(*~
	<docu>
		<summary>
			Provides dialog with the user to allow for deciding how to proceed in case of failure.	
		</summary>	
	</docu>	
~*)
FUNCTION_BLOCK PUBLIC TcoInspectorDialog EXTENDS TcoCore.TcoDialogBase
VAR
    _dialogRetry : BOOL;
    _dialogTerminate : BOOL;
    _dialogOverride : BOOL;
    _dialogIsClosed : BOOL;
    _isOverInspected : BOOL;
    {attribute 'hide'}
    _refInspector : REFERENCE TO TcoInspector;
    {attribute 'hide'}
    _tierAct : TcoCore.TcoTier(THIS^);

    _rTrigRetry : R_TRIG;
    _rTrigTerminate : R_TRIG;
    _externalCloseReq : BOOL;
    _closeRetrySignal : BOOL;
    _closeTerminateSignal : BOOL;

    _instruction : STRING(255);
    _source : STRING(255);
    _imageHeight : REAL;
    _imageWidth : REAL;
    _hideOverideButton : BOOL;
    _hideTerminateButton : BOOL;
    _hideRetryButton : BOOL;

    _showFailureDescription : BOOL;
    _showErrorCode : BOOL;
    _showDescription : BOOL;

    _isInvoked : BOOL;
END_VAR

SUPER^();

PROPERTY DialogIsClosed: REFERENCE TO BOOL
GET
DialogIsClosed ref=_dialogIsClosed;
END_GET
END_PROPERTY

PROPERTY DialogOverride: REFERENCE TO BOOL
GET
DialogOverride ref=_dialogOverride;
END_GET
END_PROPERTY

PROPERTY DialogRetry: REFERENCE TO BOOL
GET
DialogRetry ref=_dialogRetry;
END_GET
END_PROPERTY

PROPERTY DialogTerminate: REFERENCE TO BOOL
GET
DialogTerminate ref=_dialogTerminate;
END_GET
END_PROPERTY

{attribute 'hide'}
METHOD PUBLIC FB_init : BOOL
VAR_INPUT
	bInitRetains : BOOL; // if TRUE, the retain variables are initialized (warm start / cold start)
	bInCopyCode : BOOL;  // if TRUE, the instance afterwards gets moved into the copy code (online change)
	ParentObject : ITcoObject;
END_VAR
END_METHOD

METHOD HandleExternalSignals
VAR_INPUT
	inRetrySignal:BOOL;
	inTerminateSignal : BOOL;
	
END_VAR

_closeRetrySignal:=FALSE;
_closeTerminateSignal:=FALSE;


_rTrigRetry(CLK:=inRetrySignal);
IF _rTrigRetry.q THEN
	_closeRetrySignal:=TRUE;
END_IF

_rTrigTerminate(CLK:=inTerminateSignal);
IF _rTrigTerminate.q THEN
	_closeTerminateSignal:=TRUE;
END_IF

 IF(_refInspector.Done) THEN	
	 	IF NOT ( _dialogRetry) THEN
			_dialogRetry:=_closeRetrySignal;
		END_IF;
		IF NOT ( _dialogTerminate) THEN
			_dialogTerminate:=_closeTerminateSignal;
		END_IF;
 END_IF
END_METHOD

PROPERTY HideOverride: REFERENCE TO BOOL
GET
HideOverride ref=_hideOverideButton;
END_GET
END_PROPERTY

PROPERTY HideRetry: REFERENCE TO BOOL
GET
HideRetry ref=_hideRetryButton;
END_GET
END_PROPERTY

PROPERTY HideTetminate: REFERENCE TO BOOL
GET
HideTetminate ref=_hideTerminateButton;
END_GET
END_PROPERTY

METHOD PROTECTED OnStart
SUPER^.OnStart();
_isInvoked:=TRUE;
_dialogIsClosed:=FALSE;
_dialogRetry	    :=  FALSE;	
_dialogTerminate  	:=  FALSE;	
_dialogOverride   	:=  FALSE;
END_METHOD

PROPERTY INTERNAL OverInspected : BOOL
GET
OverInspected := _isOverInspected;
END_GET
SET
_isOverInspected := OverInspected;
END_SET
END_PROPERTY

METHOD Restore : TcoCore.ITcoRestorable
VAR_INPUT
END_VAR
SUPER^.Restore();
_dialogRetry	    :=  FALSE;	
_dialogTerminate  	:=  FALSE;	
_dialogOverride   	:=  FALSE;

_instruction:='';
_source:='';
_hideOverideButton:=FALSE;
_hideRetryButton:=FALSE;
_hideTerminateButton:=FALSE;
_imageHeight:=400;
_imageWidth:=600;
_showDescription:=FALSE;
_showFailureDescription:=FALSE;
_showErrorCode:=FALSE;
_isInvoked:=FALSE;
END_METHOD

METHOD SetImageSource
VAR_INPUT
	inSource:STRING(255);
	inHeight:REAL;
	inWidth:REAL;
END_VAR
_source:=inSource;
_imageHeight:=inHeight;
_imageWidth:= inWidth;
END_METHOD

METHOD SetInspector
VAR_INPUT 
	refInspector : REFERENCE TO TcoInspector;
END_VAR
_refInspector REF= refInspector;
END_METHOD

METHOD SetInstruction
VAR_INPUT
	inInstruction:STRING(255);
END_VAR
_instruction:=inInstruction;
END_METHOD

METHOD Show
VAR_INPUT
	inRetryStep : INT;
END_VAR
_isOverInspected := _refInspector.OverInspected;

IF(_tierAct.IsNewTier()) THEN
	THIS^.Restore();
END_IF

 IF(_refInspector.Done) THEN		
	IF(_refInspector.Result = eInspectorResult.Failed) THEN
		THIS^.Invoke();
		SUPER^();	
		{warning disable C0357}
		IF(_dialogRetry AND _dialogIsClosed) THEN
			_isInvoked:=FALSE;
			_refInspector.Retry(inRetryStep);
		END_IF
		
		IF(_dialogTerminate AND _dialogIsClosed) THEN
			_isInvoked:=FALSE;
			_refInspector.Terminate();
		END_IF
		
		IF(_dialogOverride AND _dialogIsClosed) THEN
			_isInvoked:=FALSE;
			_refInspector.CarryOn();
		END_IF
		{warning enable C0357}
	ELSE
		IF(_refInspector.Coordinator <> 0) THEN
			_refInspector.Coordinator.MoveNext();
		END_IF;	
	END_IF;	
END_IF;

IF THIS^._taskState=eTaskState.Done 
		AND ( _dialogRetry
		OR _dialogTerminate
		OR _dialogOverride)
		and _dialogIsClosed  THEN	
	THIS^.Restore();
END_IF;
END_METHOD

PROPERTY ShowDescription: REFERENCE TO BOOL
GET
ShowDescription ref=_showDescription;
END_GET
END_PROPERTY

PROPERTY ShowErrorCode: REFERENCE TO BOOL
GET
ShowErrorCode ref=_showErrorCode;
END_GET
END_PROPERTY

PROPERTY ShowFailureDescription: REFERENCE TO BOOL
GET
ShowFailureDescription ref=_showFailureDescription;
END_GET
END_PROPERTY

METHOD ShowWithExternalClose
VAR_INPUT
	inRetryStep : INT;
	inRetrySignal:BOOL;
	inTerminateSignal : BOOL;
	
END_VAR
//IF THIS^._taskState=eTaskState.Ready THEN
//	_dialogRetry	    	:=  FALSE;	
//	_dialogTerminate  	:=  FALSE;	
//	_dialogOverride   	:=  FALSE;
//END_IF

_isOverInspected := _refInspector.OverInspected;

IF(_tierAct.IsNewTier()) THEN
	THIS^.Restore();
END_IF

HandleExternalSignals(inRetrySignal:=inRetrySignal,inTerminateSignal:=inTerminateSignal);


 IF(_refInspector.Done) THEN		
	IF(_refInspector.Result = eInspectorResult.Failed) THEN
		THIS^.Invoke();
		SUPER^();	
		{warning disable C0357}
		//retry
	
		
		IF(_dialogRetry AND _dialogIsClosed) THEN
			_isInvoked:=FALSE;
			_refInspector.Retry(inRetryStep);
		END_IF
		//terminate
		
		IF(_dialogTerminate  AND  _dialogIsClosed) THEN
			_isInvoked:=FALSE;
			_refInspector.Terminate();
		END_IF
		
		IF(_dialogOverride AND _dialogIsClosed) THEN
			_isInvoked:=FALSE;
			_refInspector.CarryOn();
		END_IF
		{warning enable C0357}
	ELSE
		IF(_refInspector.Coordinator <> 0) THEN
			_refInspector.Coordinator.MoveNext();
		END_IF;	
	END_IF;	
END_IF;


IF THIS^._taskState=eTaskState.Done 
		AND ( _dialogRetry
		OR _dialogTerminate
		OR _dialogOverride)
		and _dialogIsClosed  THEN	
	THIS^.Restore();
END_IF;
END_METHOD

END_FUNCTION_BLOCK

(* stored: Version 1.1.0.1, ProductVersion 3.1.4024.12
   POU TcoInspectorDialog: Id {c6c9fa75-2ded-0851-0bf8-095f61987545}, SpecialFunc None
   Folder HideButtons: Id {fc417521-ac0f-06c0-055c-823e05cd5e84}
   Property DialogIsClosed: Id {900abfef-1a0b-0cce-18b4-df02c0b16f5f}
   Get Get: Id {5e312fda-6cce-064e-0243-b8216abdd75e}
   Property DialogOverride: Id {281b3990-8d8d-0186-31f8-bf848fda4f1c}
   Get Get: Id {95830134-ead6-01d5-1f16-0598f3037cba}
   Property DialogRetry: Id {dfa7c167-d55b-0582-151b-0d52ee730a93}
   Get Get: Id {c89bbf42-f18d-01a7-2d2c-1e07d87b2852}
   Property DialogTerminate: Id {4fa1d0b1-f38a-01a5-29f5-3a702c142068}
   Get Get: Id {42cb2924-62bf-0436-3801-068fa1c81f9c}
   Method FB_init: Id {1eeabd82-0765-01f0-1e37-da5161467ea2}
   Method HandleExternalSignals: Id {14a31570-9b7f-0461-2846-3d69314473d6}
   Property HideOverride: Id {84ae2f9c-a4d8-020b-3781-7d312f950a67}
   Get Get: Id {cb6df88c-aa6e-0895-0f52-62a83a5f7339}
   Property HideRetry: Id {0451d871-1284-0eba-21d9-f2d59ebaaa76}
   Get Get: Id {4cd12cda-7c87-079c-3625-1a9834368f28}
   Property HideTetminate: Id {28b62800-6c31-0d8a-222a-9e251ae995de}
   Get Get: Id {eeefe351-e74d-0f82-16d2-250018ec86f3}
   Method OnStart: Id {4e966f6d-76df-011e-1b96-699bb030acd0}
   Property OverInspected: Id {c039d7c8-ebe8-06e7-0a4c-2c6e9d3b65b1}
   Get Get: Id {2cff58c9-26c6-058e-2a22-8b77b31102ff}
   Set Set: Id {afe25584-5d3b-06f4-2804-c454f9d136dc}
   Method Restore: Id {f6a8b19c-7de2-0d61-29e8-f9ef96a63093}
   Method SetImageSource: Id {eb1ebace-4d18-04ce-12df-a38f92f39585}
   Method SetInspector: Id {59f6bb8e-40b5-01f0-1137-0e38be5ca644}
   Method SetInstruction: Id {a27a8031-8f15-094c-1f76-4c697b319fbf}
   Method Show: Id {409527dd-7ec4-05bd-0a53-372d7df86c62}
   Property ShowDescription: Id {04301ae4-3bbf-01b9-0f26-429a5fcb5a78}
   Get Get: Id {aba9d6bb-2ed1-0d20-0c13-83ac210d5219}
   Property ShowErrorCode: Id {5d0895ac-ac37-05c8-0546-600355d053f3}
   Get Get: Id {7963a26b-1d4b-01ec-2f04-af4b01ee12ef}
   Property ShowFailureDescription: Id {388439b9-2b0d-035a-3ccf-e519ea25639f}
   Get Get: Id {4023948d-09d9-0a1a-36d7-38282c54ea38}
   Method ShowWithExternalClose: Id {e354156d-00e4-0400-3d3e-1803329c2fbb} *)
